(* CoDeSys 2.3.5.6 project: kostrzewa_03.pro *)
(* Libraries: Standard.lib*4.1.15 16:23:13, SYSLIBCALLBACK.LIB*4.1.15 16:23:13 *)

(* PLC configuration (modules and I/O channels)
Configuration EC4P-200 [Root] node -1, in %IB0 out %QB0 {EC4P_RestartPwrOn = WARMSTART; EC4P_MaxCycleTime = 20; EC4P_Com1BaudRate = 38400; EC4P_CAN1BaudRate = 125KBaud; EC4P_RoutingId = 127; EC4P_EasyNetId = 1; EC4P_EasyNetCfg = 0; EC4P_EasyNetCycleTime = 50; EC4P_RoutingChannel = CAN1; EC4P_IPFlags = 0; EC4P_IPAddress = 0; EC4P_SubNetMask = 0; EC4P_DefaultGateway = 0; EC4P_SummerWinterFlags = 0; EC4P_SummerWinterRule1 = 0; EC4P_SummerWinterRule2 = 0}
  Local I/O [EC4P_LocalIO] node 0, in %IB0 out %QB0 {EC4P_LocalInt = 0}
    I1 AT %IX0.0 [LocalBitInput] Input I1
    I2 AT %IX0.1 [LocalBitInput] Input I2
    I3 AT %IX0.2 [LocalBitInput] Input I3
    I4 AT %IX0.3 [LocalBitInput] Input I4
    I5 AT %IX0.4 [LocalBitInput] Input I5
    I6 AT %IX0.5 [LocalBitInput] Input I6
    I7 AT %IX0.6 [LocalBitInput] Input I7
    I8 AT %IX0.7 [LocalBitInput] Input I8
    I9 AT %IX1.0 [LocalBitInput] Input I9
    I10 AT %IX1.1 [LocalBitInput] Input I10
    I11 AT %IX1.2 [LocalBitInput] Input I11
    I12 AT %IX1.3 [LocalBitInput] Input I12
    I13 AT %IX1.4 [LocalDiagInput] Diagnostic Input I13
    I14 AT %IX1.5 [LocalDiagInput] Diagnostic Input I14
    I15 AT %IX1.6 [LocalDiagInput] Diagnostic Input I15
    I16 AT %IX1.7 [LocalDiagInput] Diagnostic Input I16
    I7_Analog AT %IW2 [LocalAnalogIn] Input I7, 10Bit, 0-10VDC
    I8_Analog AT %IW4 [LocalAnalogIn] Input I8, 10Bit, 0-10VDC
    I11_Analog AT %IW6 [LocalAnalogIn] Input I11, 10Bit, 0-10VDC
    I12_Analog AT %IW8 [LocalAnalogIn] Input I12, 10Bit, 0-10VDC
    Transistor Outputs [EC4P_TOutputs] node 0, in %IB10 out %QB0
      Q1 AT %QX0.0 [LocalBitOutput] Transistor-Output Q1
      Q2 AT %QX0.1 [LocalBitOutput] Transistor-Output Q2
      Q3 AT %QX0.2 [LocalBitOutput] Transistor-Output Q3
      Q4 AT %QX0.3 [LocalBitOutput] Transistor-Output Q4
      Q5 AT %QX0.4 [LocalBitOutput] Transistor-Output Q5
      Q6 AT %QX0.5 [LocalBitOutput] Transistor-Output Q6
      Q7 AT %QX0.6 [LocalBitOutput] Transistor-Output Q7
      Q8 AT %QX0.7 [LocalBitOutput] Transistor-Output Q8
    No Analog Output [EC4P_NoAnalogOutput] node 1, in %IB10 out %QB1
    No Keys [EC4P_NoKeys] node 2, in %IB10 out %QB1
    No Counter [EC4P_NoCounter] node 3, in %IB10 out %QB1
  Extension [EC4P_Extension] node 1, in %IB10 out %QB1
    No Extension [EC4P_NoExtension] node 0, in %IB10 out %QB1
*)

(* POU PLC_PRG, LD *)
PROGRAM PLC_PRG
VAR
	t1: TON;
	t2: TON;
	x1: BOOL;
	wartosc: INT;
	licznik2: CTUD;
	QD:BOOL;
	t3: TP;
	x2: BOOL;
	cu: CTU;
	y1: BOOL;
	y2: BOOL;
	w1: BOOL;
	y3: BOOL;
	TP: TP;
	reset:BOOL;
	licznik1: CTU;
	cykl: INT;


END_VAR
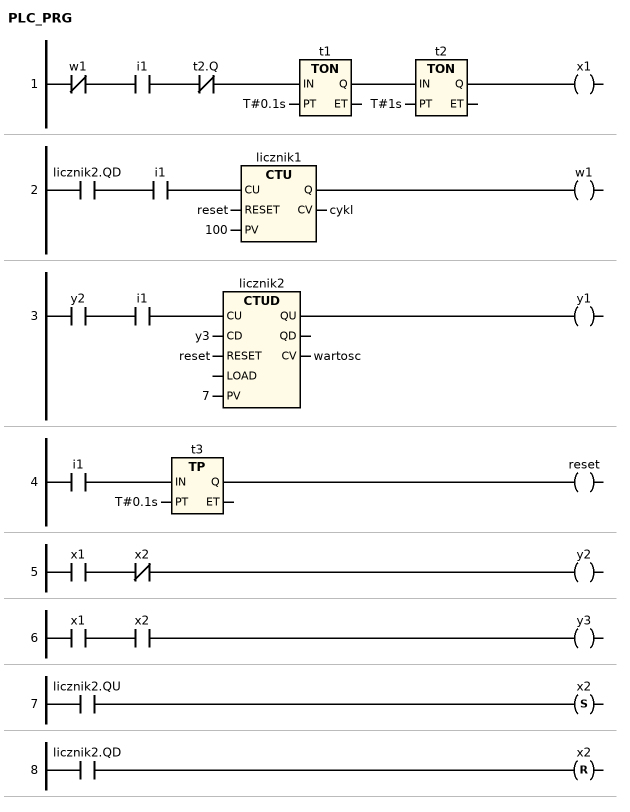
_LD_ (* Ladder Diagram *)
NETWORK 1
	[/w1] - [i1] - [/t2.Q] - t1:TON(IN: *, PT: T#0.1s) - t2:TON(IN: *, PT: T#1s) --- (x1)
NETWORK 2
	[licznik2.QD] - [i1] - licznik1:CTU(CU: *, RESET: reset, PV: 100, CV => cykl) --- (w1)
NETWORK 3
	[y2] - [i1] - licznik2:CTUD(CU: *, CD: y3, RESET: reset, LOAD: , PV: 7, CV => wartosc) --- (y1)
NETWORK 4
	[i1] - t3:TP(IN: *, PT: T#0.1s) --- (reset)
NETWORK 5
	[x1] - [/x2] --- (y2)
NETWORK 6
	[x1] - [x2] --- (y3)
NETWORK 7
	[licznik2.QU] --- (S x2)
NETWORK 8
	[licznik2.QD] --- (R x2)
_END_LD_
(* the same logic as Structured Text *)
(* Network 1 *)
t1(IN := NOT w1 AND i1 AND NOT t2.Q, PT := T#0.1s);
t2(IN := t1.Q, PT := T#1s);
x1 := t2.Q;
(* Network 2 *)
licznik1(CU := licznik2.QD AND i1, RESET := reset, PV := 100);
cykl := licznik1.CV;
w1 := licznik1.Q;
(* Network 3: see the listing above *)
(* Network 4 *)
t3(IN := i1, PT := T#0.1s);
reset := t3.Q;
(* Network 5 *)
y2 := x1 AND NOT x2;
(* Network 6 *)
y3 := x1 AND x2;
(* Network 7 *)
IF licznik2.QU THEN x2 := TRUE; END_IF;
(* Network 8 *)
IF licznik2.QD THEN x2 := FALSE; END_IF;
END_PROGRAM
